// TIA Portal project "ServoPLS 171224" (V19)

(* hardware
DEVICE "S7-1200 station_1"  S7-1200 Station
   slot 0: "Rack_0"  S7-1200 Rack  Rack  V1.0
   slot 1: "PLC_1"  CPU 1214C AC/DC/Rly  6ES7 214-1BG40-0XB0  V4.4
   slot 2: "DI 8x24VDC/DQ 8xRelay_1"  SM 1223 DI8/DQ8 x relay  6ES7 223-1PH32-0XB0  V2.0
   slot 3: "AQ 1x12BIT_1"  AQ1 signal board  6ES7 232-4HA30-0XB0  V1.0
DEVICE "SINAMICS V_1"  SINAMICS V
   slot 0: "SINAMICS V90 PN Rack"  Rail  1.0
   slot 0: "Drive_1"  V90 PN  6SL3 210-5FB10-4UFx  V1.5
      slot 1: "Drive object"  Drive Object
         slot 1: "Module access point"  Module Access Point
         slot 2: "Without PROFIsafe"  No ProfiSafe
         slot 3: "Telegram"  Standard Telegramm 3
*)

// ===== PLC "PLC_1"  CPU 1214C AC/DC/Rly =====

VAR_GLOBAL   // PLC tag table "Default tag table"
   "Axis_1_Drive_IN" AT %I68.0 : "PD_TEL3_IN";
   "Axis_1_Drive_OUT" AT %Q82.0 : "PD_TEL3_OUT";
   "Axis_1_Homing switch" AT %I0.3 : Bool;
   "firstscan" AT %M10.0 : Bool;
   "Homing procedure" AT %M11.0 : Bool;
   "Home_Done_Vertical" AT %M11.1 : Bool;
   "Tag_1" AT %I2.0 : Bool;
   "Tag_2" AT %M20.0 : Bool;
   "ServoONHorizont" AT %Q0.7 : Bool;
   "home_horizontal" AT %Q0.4 : Bool;
   "Home_done_horizontal" AT %M12.0 : Bool;
   "HomeComplete" AT %I8.0 : Bool;
   "Tag_3" AT %I1.3 : Bool;
   "Servo_fault" AT %I1.4 : Bool;
   "Servo_Alarm" AT %I1.5 : Bool;
   "Tag_4" AT %M100.0 : Bool;
   "System_Byte" AT %MB8001 : Byte;
   "FirstScan(1)" AT %M1.0 : Bool;
   "DiagStatusUpdate" AT %M8001.1 : Bool;
   "AlwaysTRUE" AT %M8001.2 : Bool;
   "AlwaysFALSE" AT %M8001.3 : Bool;
   "Clock_Byte" AT %MB8000 : Byte;
   "Clock_10Hz" AT %M8000.0 : Bool;
   "Clock_5Hz" AT %M8000.1 : Bool;
   "Clock_2.5Hz" AT %M8000.2 : Bool;
   "Clock_2Hz" AT %M8000.3 : Bool;
   "Clock_1.25Hz" AT %M8000.4 : Bool;
   "Clock_1Hz" AT %M8000.5 : Bool;
   "Clock_0.625Hz" AT %M8000.6 : Bool;
   "Clock_0.5Hz" AT %M8000.7 : Bool;
   "Tag_5" AT %M100.1 : Bool;
   "Reset_HorizontDrive" AT %Q0.6 : Bool;
   "hent 8cm" AT %M1000.0 : Bool;
   "Binær_hent_8cm" AT %M50.0 : Bool;
   "Stepdata_1_U" AT %Q0.1 : Bool;
   "Stepdata_2_U" AT %Q0.2 : Bool;
   "Stepdata_3_U" AT %Q0.3 : Bool;
   "Stepdata_1_Conf" AT %I0.6 : Bool;
   "Stepdata_2_Conf" AT %I0.7 : Bool;
   "Stepdata_3_Conf" AT %I1.0 : Bool;
   "Drive_Servo" AT %Q0.5 : Bool;
   "lever_8cm" AT %M1000.1 : Bool;
   "binær _lever_8cm" AT %M50.1 : Bool;
   "Sett sylinder C7" AT %M50.7 : Bool;
   "Sylinder C7" AT %Q0.0 : Bool;
   "Tag_8" AT %M50.2 : Bool;
   "Hent_16cm" AT %M50.4 : Bool;
   "Binær_Hent_16cm" AT %M50.5 : Bool;
   "Lever_16cm" AT %M50.6 : Bool;
   "binær_lever_16cm" AT %M51.0 : Bool;
   "Hent_8cm_fra_main" AT %I0.0 : Bool;
   "Lever_8cm_fra_Main" AT %I8.1 : Bool;
   "Servo_går" AT %I1.1 : Bool;
   "Klar_for_pall_8cm" AT %Q8.0 : Bool;
   "Klar_for_pall_12cm" AT %Q8.1 : Bool;
   "Servo_INP" AT %I1.2 : Bool;
   "Tag_6" AT %M200.0 : Bool;
   "Tag_7" AT %M200.1 : Bool;
   "Tag_9" AT %M200.2 : Bool;
   "Tag_10" AT %M200.3 : Bool;
   "Tag_11" AT %M201.0 : Bool;
   "C7_Retur_Set_8cm" AT %M2.0 : Bool;
   "C7_min_pos" AT %I0.4 : Bool;
   "c7_pluss_pos" AT %I0.5 : Bool;
   "Bekreftet_levering_8cm" AT %Q2.4 : Bool;
   "Bekreftet_levering_8cm_NYY" AT %Q8.4 : Bool;
   "Klar_for_pall_16cm" AT %Q8.2 : Bool;
   "Lever_12cm_fra_main" AT %I8.2 : Bool;
   "Lever_16cm_fra_main" AT %I8.3 : Bool;
   "C7_retur_set_16cm" AT %M3.0 : Bool;
   "Bekreftet_levering_16cm_NYY" AT %Q8.6 : Bool;
   "Hent_16cm_fra_main" AT %I0.2 : Bool;
   "Sett_leveringsposisjon_Horizont_Unngå_Hylle" AT %M210.0 : Bool;
   "Tag_13" AT %M210.1 : Bool;
   "Sett_Sylinder_C7_16cm" AT %M52.0 : Bool;
   "Binær_Hent_12cm" AT %M51.1 : Bool;
   "Hent_12cm_fra_main" AT %I0.1 : Bool;
   "Binær_lever_12cm" AT %M51.2 : Bool;
   "C7_retur_set_12cm" AT %M3.1 : Bool;
   "Sett_Sylinder_C7_12cm" AT %M52.1 : Bool;
   "Bekreftet_levering_12cm_NYY" AT %Q8.5 : Bool;
   "Tag_12" AT %M211.0 : Bool;
   "Forrigling_c7_8cm" AT %M111.0 : Bool;
   "Forrigling_c7_16cm" AT %M111.1 : Bool;
   "Forrigling_c7_12cm" AT %M111.2 : Bool;
END_VAR

// folder: System blocks/Program resources

DATA_BLOCK "IEC_Timer_0_DB"   // DB4
{ S7_Optimized_Access := 'TRUE' }
AUTHOR : Simatic
FAMILY : IEC
NAME : IEC_TMR
VERSION : 1.0
// stored: InstanceOfName IEC_TIMER
"IEC_TIMER"
BEGIN
END_DATA_BLOCK

DATA_BLOCK "ton 8cm enable move absolute"   // DB5
{ S7_Optimized_Access := 'TRUE' }
AUTHOR : Simatic
FAMILY : IEC
NAME : IEC_TMR
VERSION : 1.0
// stored: InstanceOfName IEC_TIMER
"IEC_TIMER"
BEGIN
END_DATA_BLOCK

DATA_BLOCK "IEC_Timer_0_DB_1"   // DB6
{ S7_Optimized_Access := 'TRUE' }
AUTHOR : Simatic
FAMILY : IEC
NAME : IEC_TMR
VERSION : 1.0
// stored: InstanceOfName IEC_TIMER
"IEC_TIMER"
BEGIN
END_DATA_BLOCK

DATA_BLOCK "delay utskyt 8cm"   // DB8
{ S7_Optimized_Access := 'TRUE' }
AUTHOR : Simatic
FAMILY : IEC
NAME : IEC_TMR
VERSION : 1.0
// stored: InstanceOfName IEC_TIMER
"IEC_TIMER"
BEGIN
END_DATA_BLOCK

DATA_BLOCK "test"   // DB10
{ S7_Optimized_Access := 'TRUE' }
AUTHOR : Simatic
FAMILY : IEC
NAME : IEC_TMR
VERSION : 1.0
// stored: InstanceOfName IEC_TIMER
"IEC_TIMER"
BEGIN
END_DATA_BLOCK

DATA_BLOCK "Timer_16cm_hent_200ms"   // DB12
{ S7_Optimized_Access := 'TRUE' }
AUTHOR : Simatic
FAMILY : IEC
NAME : IEC_TMR
VERSION : 1.0
// stored: InstanceOfName IEC_TIMER
"IEC_TIMER"
BEGIN
END_DATA_BLOCK

DATA_BLOCK "testing"   // DB14
{ S7_Optimized_Access := 'TRUE' }
AUTHOR : Simatic
FAMILY : IEC
NAME : IEC_TMR
VERSION : 1.0
// stored: InstanceOfName IEC_TIMER
"IEC_TIMER"
BEGIN
END_DATA_BLOCK

DATA_BLOCK "IEC_Timer_0_DB_2"   // DB15
{ S7_Optimized_Access := 'TRUE' }
AUTHOR : Simatic
FAMILY : IEC
NAME : IEC_TMR
VERSION : 1.0
// stored: InstanceOfName IEC_TIMER
"IEC_TIMER"
BEGIN
END_DATA_BLOCK

DATA_BLOCK "IEC_Timer_0_DB_3"   // DB16
{ S7_Optimized_Access := 'TRUE' }
AUTHOR : Simatic
FAMILY : IEC
NAME : IEC_TMR
VERSION : 1.0
// stored: InstanceOfName IEC_TIMER
"IEC_TIMER"
BEGIN
END_DATA_BLOCK

DATA_BLOCK "test10"   // DB17
{ S7_Optimized_Access := 'TRUE' }
AUTHOR : Simatic
FAMILY : IEC
NAME : IEC_TMR
VERSION : 1.0
// stored: InstanceOfName IEC_TIMER
"IEC_TIMER"
BEGIN
END_DATA_BLOCK

DATA_BLOCK "Hent_12cm_Delay_200ms"   // DB18
{ S7_Optimized_Access := 'TRUE' }
AUTHOR : Simatic
FAMILY : IEC
NAME : IEC_TMR
VERSION : 1.0
// stored: InstanceOfName IEC_TIMER
"IEC_TIMER"
BEGIN
END_DATA_BLOCK

DATA_BLOCK "Delay_utskyt_12cm"   // DB21
{ S7_Optimized_Access := 'TRUE' }
AUTHOR : Simatic
FAMILY : IEC
NAME : IEC_TMR
VERSION : 1.0
// stored: InstanceOfName IEC_TIMER
"IEC_TIMER"
BEGIN
END_DATA_BLOCK

DATA_BLOCK "TP_Bekreft_Levering_12cm"   // DB22
{ S7_Optimized_Access := 'TRUE' }
AUTHOR : Simatic
FAMILY : IEC
NAME : IEC_TMR
VERSION : 1.0
// stored: InstanceOfName IEC_TIMER
"IEC_TIMER"
BEGIN
END_DATA_BLOCK

// folder: (top level)

DATA_BLOCK "Axis_1"   // DB1, Motion_DB
{ S7_Optimized_Access := 'TRUE' }
AUTHOR : SIMATIC
FAMILY : BasicMC
NAME : TO_PosAx
VERSION : 7.0
// stored: InstanceOfName TO_PositioningAxis
"TO_PositioningAxis"
BEGIN
   // Axis.HomingReferencePointSwitch_AddressCU = %I0.3
   // Axis.Encoder.OfflineDataAdaption = TRUE
   // Axis.Encoder.TelegramAddressOutCU = %Q82.0
   // Axis.Encoder.TelegramAddressInCU = %I68.0
   // Axis.Encoder.DoNameCU = Drive_1.Drive object_Encoder1
   // Axis.Drive.OfflineDataAdaption = TRUE
   // Axis.Drive.TelegramAddressOutCU = %Q82.0
   // Axis.Drive.TelegramAddressInCU = %I68.0
   // Axis.Drive.TelegramType = 2
   // Axis.Drive.DoNameCU = Drive_1.Drive object
   // Axis.LengthUnitNormalized.Time = 1
   // Axis.LengthUnitNormalized.Distance = -2
   // Axis.Encoder.SelectedHscIndexCU = -1
   // Axis.Encoder.DbTypeCU = Classic
   // Axis.Drive.DbTypeCU = Classic
END_DATA_BLOCK

FUNCTION "Utgangssignaler" : Void   // FC1, LAD
{ S7_Optimized_Access := 'TRUE' }
VERSION : 0.1
   VAR_TEMP   // added for the SCL form of the ladder/FBD networks
      _w1 : Bool;
   END_VAR
BEGIN

REGION Network 1: Utganger Horizont_servo + syl
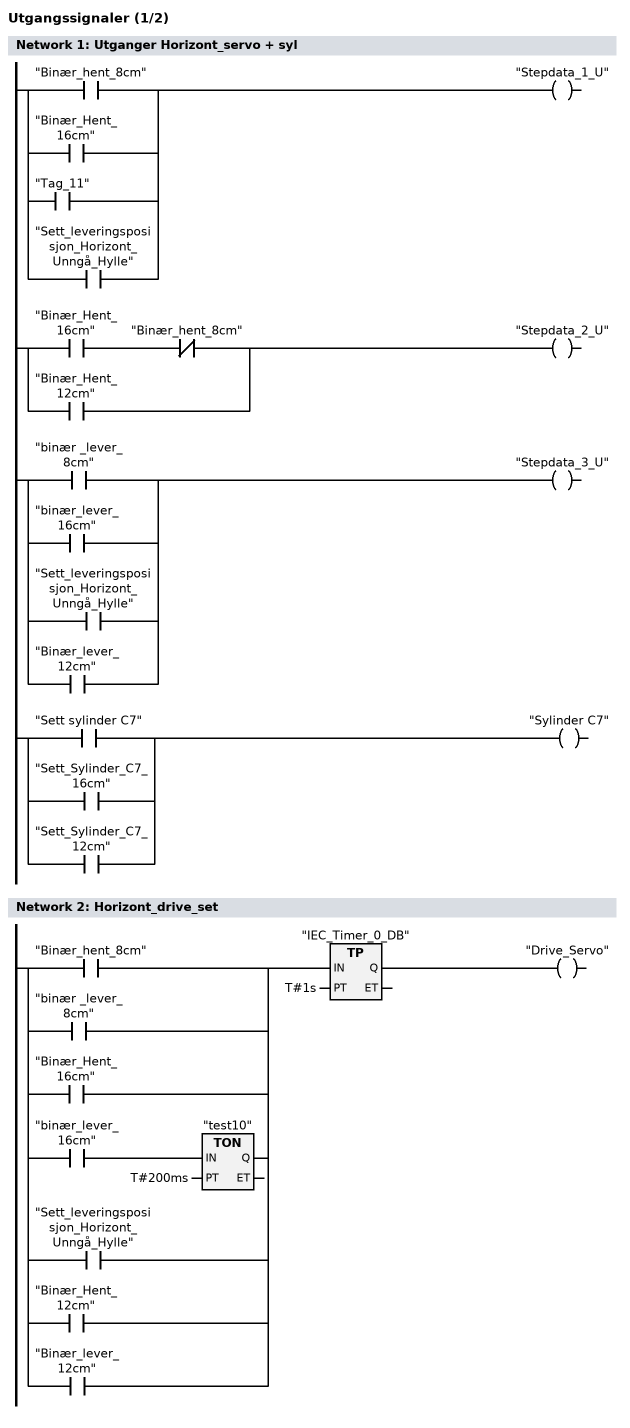
   RUNG wire#powerrail
      Contact( "Binær_hent_8cm" )
      wire#w1
      Coil( "Stepdata_1_U" )
   END_RUNG
   RUNG wire#powerrail
      Contact( "Binær_Hent_16cm" )
   END_RUNG wire#w1
   RUNG wire#powerrail
      Contact( "Tag_11" )
   END_RUNG wire#w1
   RUNG wire#powerrail
      Contact( "Sett_leveringsposisjon_Horizont_Unngå_Hylle" )
   END_RUNG wire#w1
   RUNG wire#powerrail
      Contact( "Binær_Hent_16cm" )
      I_Contact( "Binær_hent_8cm" )
      wire#w2
      Coil( "Stepdata_2_U" )
   END_RUNG
   RUNG wire#powerrail
      Contact( "Binær_Hent_12cm" )
   END_RUNG wire#w2
   RUNG wire#powerrail
      Contact( "binær _lever_8cm" )
      wire#w3
      Coil( "Stepdata_3_U" )
   END_RUNG
   RUNG wire#powerrail
      Contact( "binær_lever_16cm" )
   END_RUNG wire#w3
   RUNG wire#powerrail
      Contact( "Sett_leveringsposisjon_Horizont_Unngå_Hylle" )
   END_RUNG wire#w3
   RUNG wire#powerrail
      Contact( "Binær_lever_12cm" )
   END_RUNG wire#w3
   RUNG wire#powerrail
      Contact( "Sett sylinder C7" )
      wire#w4
      Coil( "Sylinder C7" )
   END_RUNG
   RUNG wire#powerrail
      Contact( "Sett_Sylinder_C7_16cm" )
   END_RUNG wire#w4
   RUNG wire#powerrail
      Contact( "Sett_Sylinder_C7_12cm" )
   END_RUNG wire#w4
   // the same network as SCL:
   "Stepdata_1_U" := "Binær_hent_8cm" OR "Binær_Hent_16cm" OR "Tag_11" OR "Sett_leveringsposisjon_Horizont_Unngå_Hylle";
   "Stepdata_2_U" := ("Binær_Hent_16cm" AND NOT "Binær_hent_8cm") OR "Binær_Hent_12cm";
   "Stepdata_3_U" := "binær _lever_8cm" OR "binær_lever_16cm" OR "Sett_leveringsposisjon_Horizont_Unngå_Hylle" OR "Binær_lever_12cm";
   "Sylinder C7" := "Sett sylinder C7" OR "Sett_Sylinder_C7_16cm" OR "Sett_Sylinder_C7_12cm";
END_REGION

REGION Network 2: Horizont_drive_set
   "test10".TON(IN := "binær_lever_16cm", PT := T#200ms);
   "IEC_Timer_0_DB".TP(IN := "Binær_hent_8cm" OR "binær _lever_8cm" OR "Binær_Hent_16cm" OR "test10".Q OR "Sett_leveringsposisjon_Horizont_Unngå_Hylle" OR "Binær_Hent_12cm" OR "Binær_lever_12cm",
                       PT := T#1s);
   "Drive_Servo" := "IEC_Timer_0_DB".Q;
END_REGION

REGION Network 3
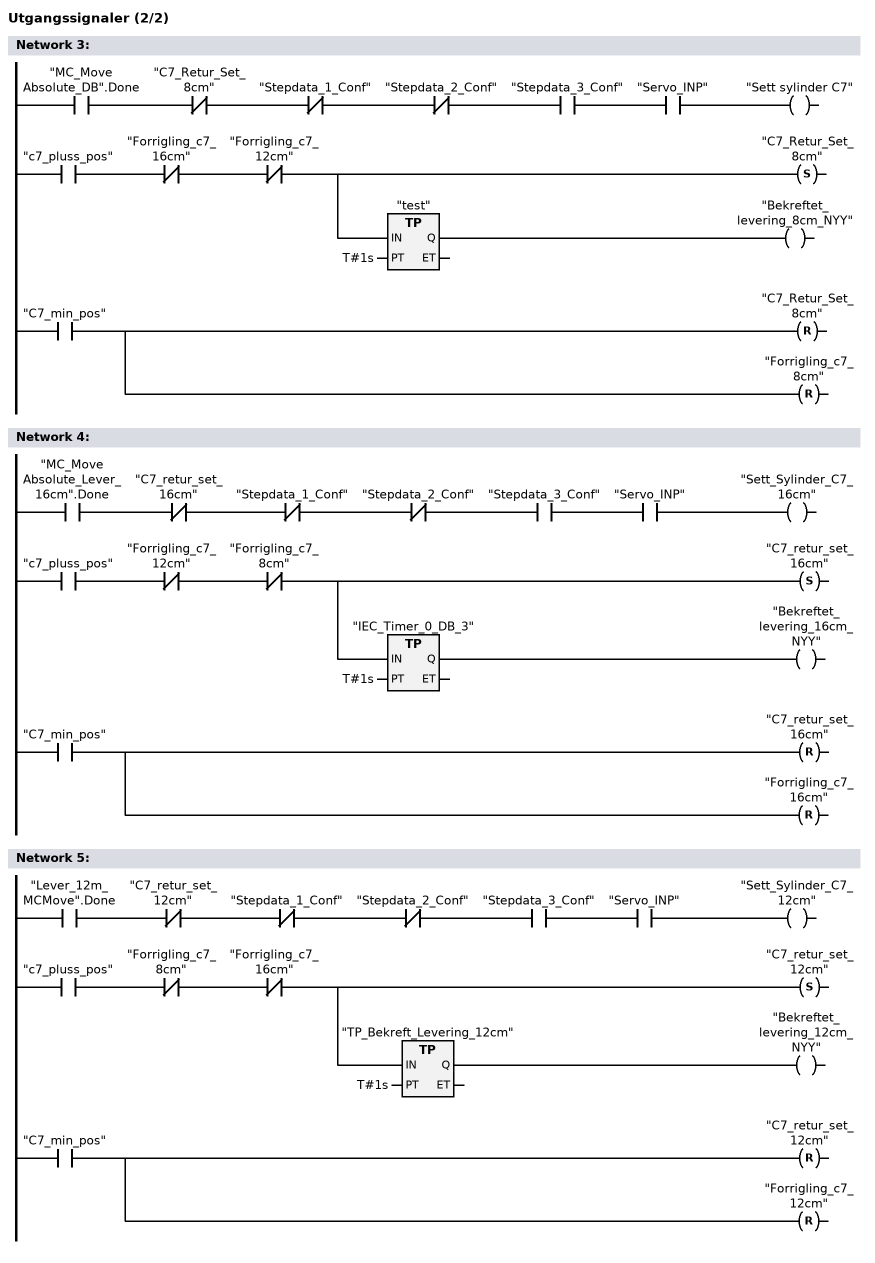
   "Sett sylinder C7" := "MC_MoveAbsolute_DB".Done AND NOT "C7_Retur_Set_8cm" AND NOT "Stepdata_1_Conf" AND NOT "Stepdata_2_Conf" AND "Stepdata_3_Conf" AND "Servo_INP";
   #_w1 := "c7_pluss_pos" AND NOT "Forrigling_c7_16cm" AND NOT "Forrigling_c7_12cm";
   IF #_w1 THEN "C7_Retur_Set_8cm" := TRUE; END_IF;
   "test".TP(IN := #_w1, PT := T#1s);
   "Bekreftet_levering_8cm_NYY" := "test".Q;
   IF "C7_min_pos" THEN
       "C7_Retur_Set_8cm" := FALSE;
       "Forrigling_c7_8cm" := FALSE;
   END_IF;
END_REGION

REGION Network 4
   "Sett_Sylinder_C7_16cm" := "MC_MoveAbsolute_Lever_16cm".Done AND NOT "C7_retur_set_16cm" AND NOT "Stepdata_1_Conf" AND NOT "Stepdata_2_Conf" AND "Stepdata_3_Conf" AND "Servo_INP";
   #_w1 := "c7_pluss_pos" AND NOT "Forrigling_c7_12cm" AND NOT "Forrigling_c7_8cm";
   IF #_w1 THEN "C7_retur_set_16cm" := TRUE; END_IF;
   "IEC_Timer_0_DB_3".TP(IN := #_w1, PT := T#1s);
   "Bekreftet_levering_16cm_NYY" := "IEC_Timer_0_DB_3".Q;
   IF "C7_min_pos" THEN
       "C7_retur_set_16cm" := FALSE;
       "Forrigling_c7_16cm" := FALSE;
   END_IF;
END_REGION

REGION Network 5
   "Sett_Sylinder_C7_12cm" := "Lever_12m_MCMove".Done AND NOT "C7_retur_set_12cm" AND NOT "Stepdata_1_Conf" AND NOT "Stepdata_2_Conf" AND "Stepdata_3_Conf" AND "Servo_INP";
   #_w1 := "c7_pluss_pos" AND NOT "Forrigling_c7_8cm" AND NOT "Forrigling_c7_16cm";
   IF #_w1 THEN "C7_retur_set_12cm" := TRUE; END_IF;
   "TP_Bekreft_Levering_12cm".TP(IN := #_w1, PT := T#1s);
   "Bekreftet_levering_12cm_NYY" := "TP_Bekreft_Levering_12cm".Q;
   IF "C7_min_pos" THEN
       "C7_retur_set_12cm" := FALSE;
       "Forrigling_c7_12cm" := FALSE;
   END_IF;
END_REGION
END_FUNCTION

FUNCTION "Posisjonering" : Void   // FC2, LAD
{ S7_Optimized_Access := 'TRUE' }
VERSION : 0.1
BEGIN

REGION Network 1: Hent 8cm
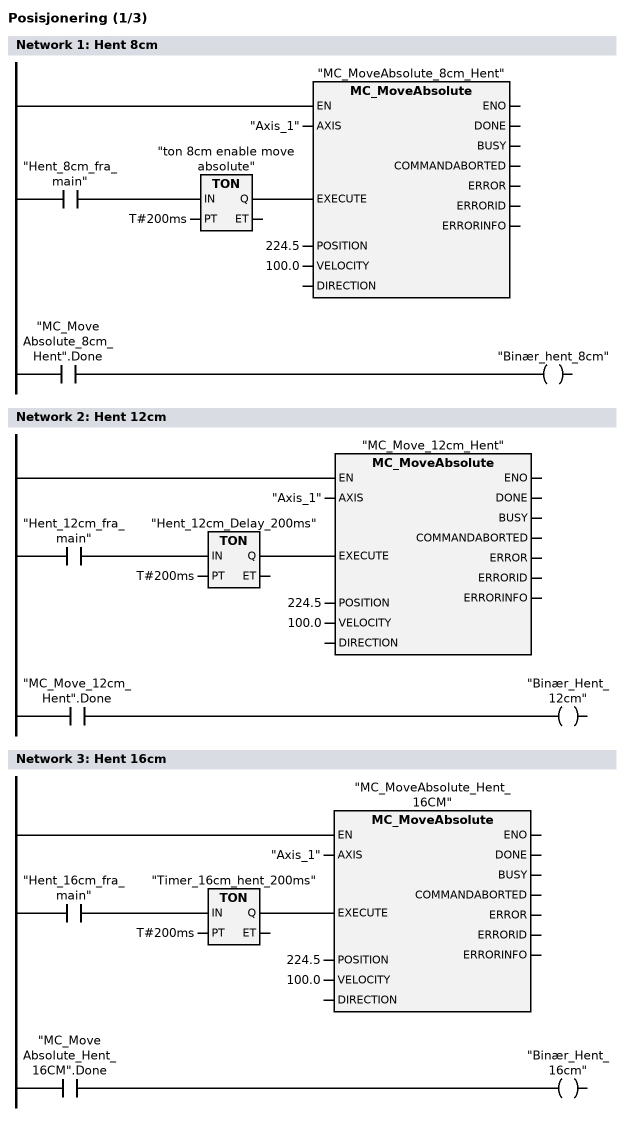
   "ton 8cm enable move absolute".TON(IN := "Hent_8cm_fra_main", PT := T#200ms);
   "MC_MoveAbsolute_8cm_Hent"(Axis := "Axis_1",   // MC_MoveAbsolute
                           Execute := "ton 8cm enable move absolute".Q,
                           Position := 224.5,
                           Velocity := 100.0);
   "Binær_hent_8cm" := "MC_MoveAbsolute_8cm_Hent".Done;
END_REGION

REGION Network 2: Hent 12cm
   "Hent_12cm_Delay_200ms".TON(IN := "Hent_12cm_fra_main", PT := T#200ms);
   "MC_Move_12cm_Hent"(Axis := "Axis_1",   // MC_MoveAbsolute
                       Execute := "Hent_12cm_Delay_200ms".Q,
                       Position := 224.5,
                       Velocity := 100.0);
   "Binær_Hent_12cm" := "MC_Move_12cm_Hent".Done;
END_REGION

REGION Network 3: Hent 16cm
   "Timer_16cm_hent_200ms".TON(IN := "Hent_16cm_fra_main", PT := T#200ms);
   "MC_MoveAbsolute_Hent_16CM"(Axis := "Axis_1",   // MC_MoveAbsolute
                           Execute := "Timer_16cm_hent_200ms".Q,
                           Position := 224.5,
                           Velocity := 100.0);
   "Binær_Hent_16cm" := "MC_MoveAbsolute_Hent_16CM".Done;
END_REGION

REGION Network 4: Lever 8cm
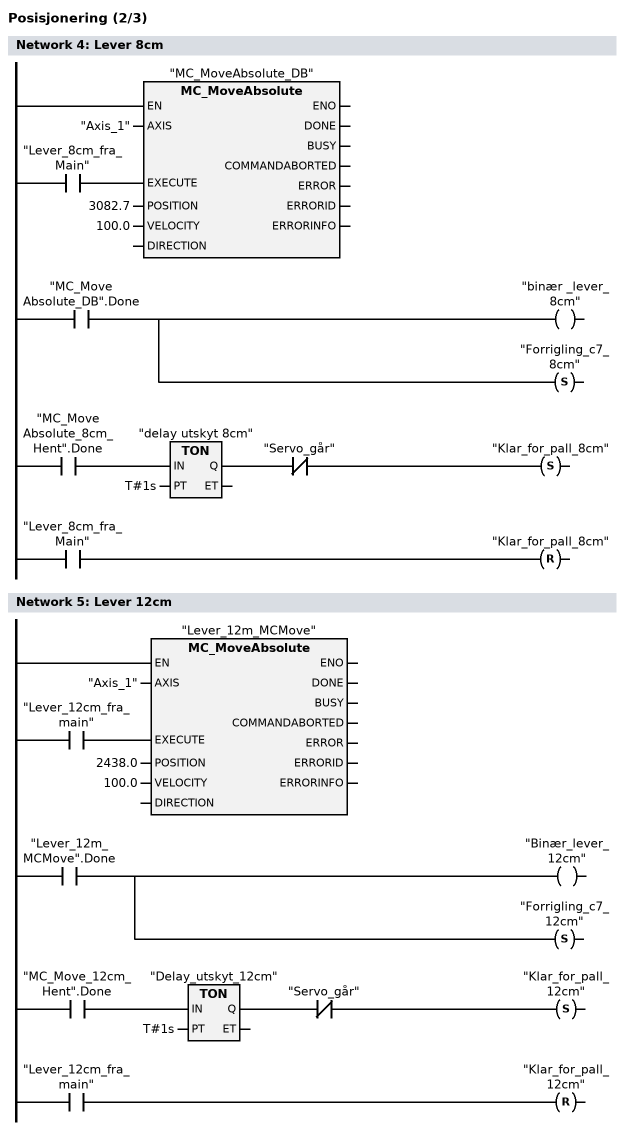
   "MC_MoveAbsolute_DB"(Axis := "Axis_1",   // MC_MoveAbsolute
                        Execute := "Lever_8cm_fra_Main",
                        Position := 3082.7,
                        Velocity := 100.0);
   "binær _lever_8cm" := "MC_MoveAbsolute_DB".Done;
   IF "MC_MoveAbsolute_DB".Done THEN "Forrigling_c7_8cm" := TRUE; END_IF;
   "delay utskyt 8cm".TON(IN := "MC_MoveAbsolute_8cm_Hent".Done, PT := T#1s);
   IF "delay utskyt 8cm".Q AND NOT "Servo_går" THEN "Klar_for_pall_8cm" := TRUE; END_IF;
   IF "Lever_8cm_fra_Main" THEN "Klar_for_pall_8cm" := FALSE; END_IF;
END_REGION

REGION Network 5: Lever 12cm
   "Lever_12m_MCMove"(Axis := "Axis_1", Execute := "Lever_12cm_fra_main", Position := 2438.0, Velocity := 100.0);   // MC_MoveAbsolute
   "Binær_lever_12cm" := "Lever_12m_MCMove".Done;
   IF "Lever_12m_MCMove".Done THEN "Forrigling_c7_12cm" := TRUE; END_IF;
   "Delay_utskyt_12cm".TON(IN := "MC_Move_12cm_Hent".Done, PT := T#1s);
   IF "Delay_utskyt_12cm".Q AND NOT "Servo_går" THEN "Klar_for_pall_12cm" := TRUE; END_IF;
   IF "Lever_12cm_fra_main" THEN "Klar_for_pall_12cm" := FALSE; END_IF;
END_REGION

REGION Network 6: Lever 16cm
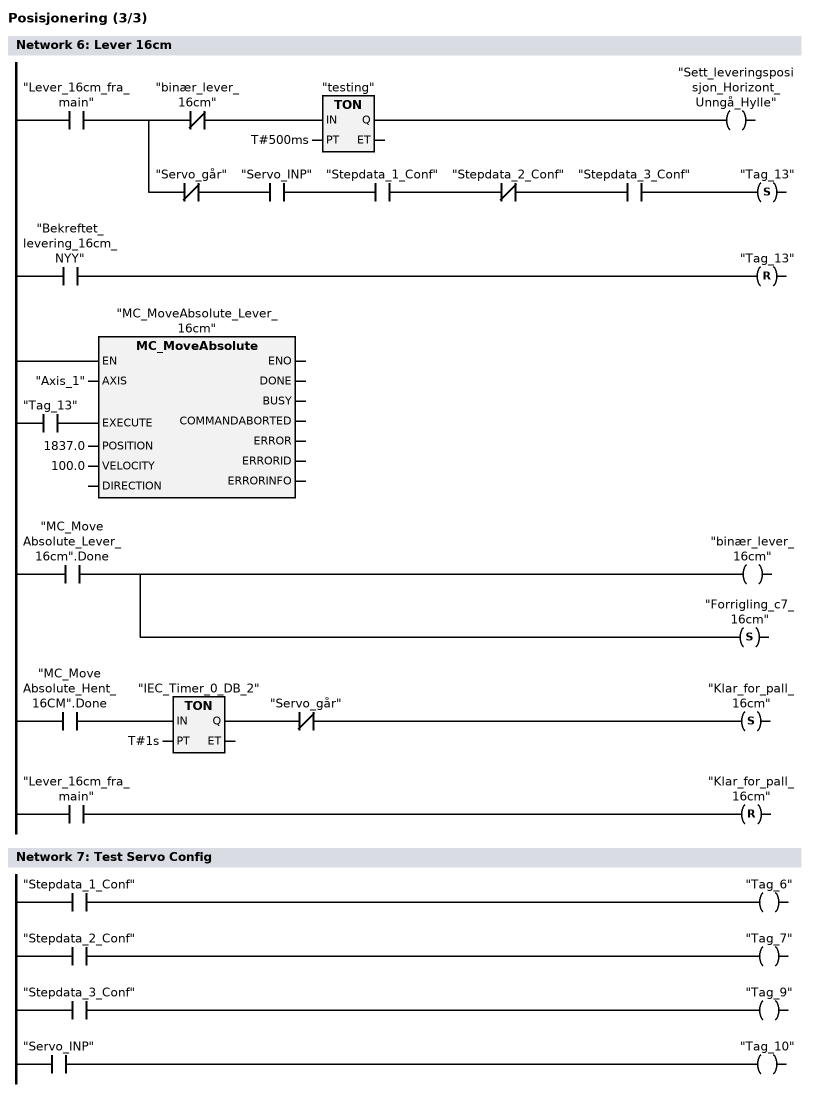
   "testing".TON(IN := "Lever_16cm_fra_main" AND NOT "binær_lever_16cm", PT := T#500ms);
   "Sett_leveringsposisjon_Horizont_Unngå_Hylle" := "testing".Q;
   IF "Lever_16cm_fra_main" AND NOT "Servo_går" AND "Servo_INP" AND "Stepdata_1_Conf" AND NOT "Stepdata_2_Conf" AND "Stepdata_3_Conf" THEN
       "Tag_13" := TRUE;
   END_IF;
   IF "Bekreftet_levering_16cm_NYY" THEN "Tag_13" := FALSE; END_IF;
   "MC_MoveAbsolute_Lever_16cm"(Axis := "Axis_1", Execute := "Tag_13", Position := 1837.0, Velocity := 100.0);   // MC_MoveAbsolute
   "binær_lever_16cm" := "MC_MoveAbsolute_Lever_16cm".Done;
   IF "MC_MoveAbsolute_Lever_16cm".Done THEN "Forrigling_c7_16cm" := TRUE; END_IF;
   "IEC_Timer_0_DB_2".TON(IN := "MC_MoveAbsolute_Hent_16CM".Done, PT := T#1s);
   IF "IEC_Timer_0_DB_2".Q AND NOT "Servo_går" THEN "Klar_for_pall_16cm" := TRUE; END_IF;
   IF "Lever_16cm_fra_main" THEN "Klar_for_pall_16cm" := FALSE; END_IF;
END_REGION

REGION Network 7: Test Servo Config
   RUNG wire#powerrail
      Contact( "Stepdata_1_Conf" )
      Coil( "Tag_6" )
   END_RUNG
   RUNG wire#powerrail
      Contact( "Stepdata_2_Conf" )
      Coil( "Tag_7" )
   END_RUNG
   RUNG wire#powerrail
      Contact( "Stepdata_3_Conf" )
      Coil( "Tag_9" )
   END_RUNG
   RUNG wire#powerrail
      Contact( "Servo_INP" )
      Coil( "Tag_10" )
   END_RUNG
   // the same network as SCL:
   "Tag_6" := "Stepdata_1_Conf";
   "Tag_7" := "Stepdata_2_Conf";
   "Tag_9" := "Stepdata_3_Conf";
   "Tag_10" := "Servo_INP";
END_REGION
END_FUNCTION

ORGANIZATION_BLOCK "Main"   // OB1, LAD, ProgramCycle
TITLE = "Main Program Sweep (Cycle)"
{ S7_Optimized_Access := 'TRUE' }
VERSION : 0.1
   VAR_INPUT
      Initial_Call : Bool;   // Initial call of this OB
      Remanence : Bool;   // =True, if remanent data are available
   END_VAR
   VAR_TEMP   // added for the SCL form of the ladder/FBD networks
      _w1 : Bool;
   END_VAR
BEGIN

REGION Network 1: Homing Vertical
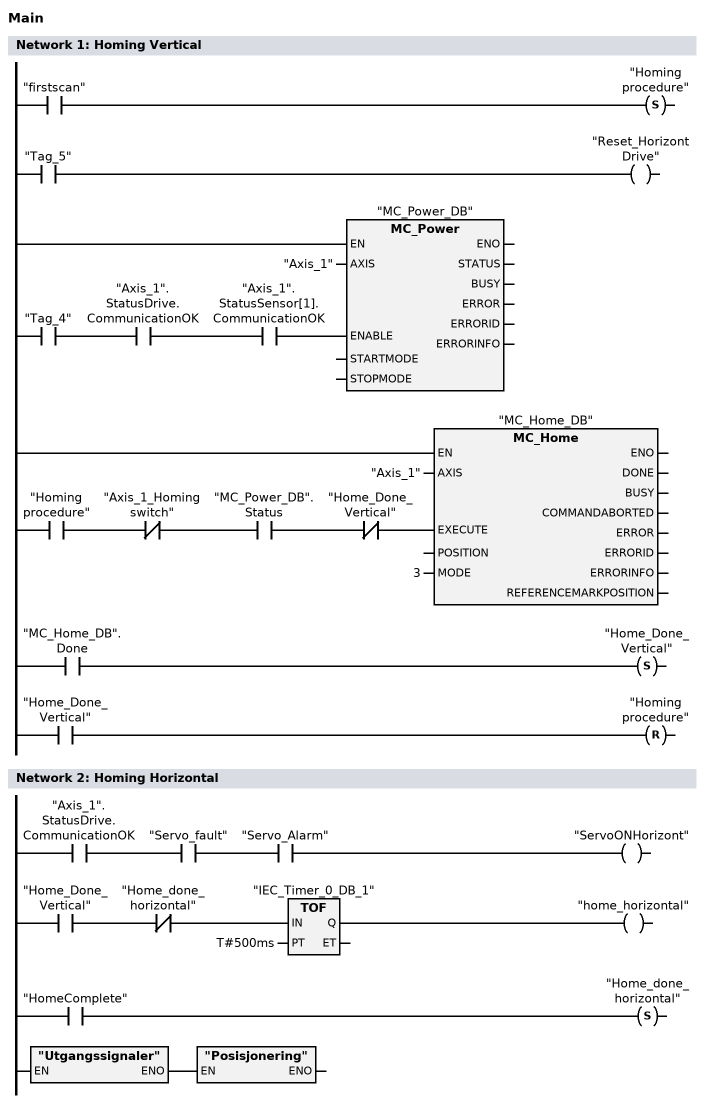
   IF "firstscan" THEN "Homing procedure" := TRUE; END_IF;
   "Reset_HorizontDrive" := "Tag_5";
   "MC_Power_DB"(Axis := "Axis_1",   // MC_Power
                 Enable := "Tag_4" AND "Axis_1".StatusDrive.CommunicationOK AND "Axis_1".StatusSensor[1].CommunicationOK);
   "MC_Home_DB"(Axis := "Axis_1",   // MC_Home
                Execute := "Homing procedure" AND NOT "Axis_1_Homing switch" AND "MC_Power_DB".Status AND NOT "Home_Done_Vertical",
                Mode := 3);
   IF "MC_Home_DB".Done THEN "Home_Done_Vertical" := TRUE; END_IF;
   IF "Home_Done_Vertical" THEN "Homing procedure" := FALSE; END_IF;
END_REGION

REGION Network 2: Homing Horizontal
   "ServoONHorizont" := "Axis_1".StatusDrive.CommunicationOK AND "Servo_fault" AND "Servo_Alarm";
   "IEC_Timer_0_DB_1".TOF(IN := "Home_Done_Vertical" AND NOT "Home_done_horizontal", PT := T#500ms);
   "home_horizontal" := "IEC_Timer_0_DB_1".Q;
   IF "HomeComplete" THEN "Home_done_horizontal" := TRUE; END_IF;
   "Utgangssignaler"(ENO => #_w1);
   IF #_w1 THEN "Posisjonering"(); END_IF;
END_REGION
END_ORGANIZATION_BLOCK